FUNCTION_BLOCK FINAL FB_Tilt_A EXTENDS FB_StatusExecuteFB
VAR_IN_OUT
	fbMover								: MC_PlanarMover;
END_VAR
VAR_INPUT
	Execute								: BOOL;
	Position							: ST_POSITION;
	Velocity							: LREAL;
	Acceleration						: LREAL;
	Deceleration						: LREAL;
	Jerk								: LREAL;
END_VAR
VAR_OUTPUT
	Done								: BOOL;
	Busy								: BOOL;
	CommandAborted						: BOOL;
	Error								: BOOL;
	ErrorID								: UDINT;
END_VAR
VAR
	uiState								: UINT;
	//Input 内部変数
	dutPosition							: ST_POSITION;
	lrVelocity							: LREAL;
	lrAcceleration						: LREAL;
	lrDeceleration						: LREAL;
	lrJerk								: LREAL;
	
	//ローカル
	fbFB_Mover							: MC_PlanarFeedback;
	dutTargetPosition					: ST_POSITION;
	fbConstraint						: DynamicConstraint_PathXY;
	fbMoveA								: FB_MoveA;
END_VAR

Prop_Execute := Execute;
METH_Main();

fbFB_Mover.Update();

Busy := bBusy;
Done := bDone;
CommandAborted := bCommandAborted;
Error := bError;
ErrorID := udiErrorID;

//{error 'add method implementation or delete method to use base implementation'}
METHOD INTERNAL METH_Busy : BOOL
IF fbFB_Mover.Error THEN
	METH_Error();
	Prop_ErrorID := fbFB_Mover.ErrorId; //Moverがエラー
	RETURN;
END_IF
IF THIS^.fbMover.MCTOPLC.STD.State = MC_PLANAR_STATE.Error THEN
	METH_Error();
	Prop_ErrorID := 1; //Moverがエラー
	RETURN;
END_IF
IF fbFB_Mover.Aborted THEN
	METH_CommandAborted();
	RETURN;
END_IF

CASE THIS^.uiState OF
	0:
	//+Aに傾ける
	dutTargetPosition.a := dutPosition.a;
	fbMoveA(
		fbMover:= THIS^.fbMover, 
		Execute:= TRUE, 
		Position:= dutTargetPosition, 
		Velocity:= THIS^.lrVelocity, 
		Acceleration:= THIS^.lrAcceleration, 
		Deceleration:= THIS^.lrDeceleration, 
		Jerk:= THIS^.lrJerk);
	IF fbMoveA.Done THEN
		fbMoveA(fbMover:= THIS^.fbMover, Execute:= FALSE);
		THIS^.uiState := 10;
	ELSIF fbMoveA.Error THEN
		METH_Error();
		Prop_ErrorID := 10; //Moverがエラー
	END_IF
	
	10:
	//-Aに傾ける
	dutTargetPosition.a := -1*dutPosition.a;
	fbMoveA(
		fbMover:= THIS^.fbMover, 
		Execute:= TRUE, 
		Position:= dutTargetPosition, 
		Velocity:= THIS^.lrVelocity, 
		Acceleration:= THIS^.lrAcceleration, 
		Deceleration:= THIS^.lrDeceleration, 
		Jerk:= THIS^.lrJerk);
	IF fbMoveA.Done THEN
		fbMoveA(fbMover:= THIS^.fbMover, Execute:= FALSE);
		THIS^.uiState := 30;
	ELSIF fbMoveA.Error THEN
		METH_Error();
		Prop_ErrorID := 11; //Moverがエラー
	END_IF

	30:
	//0に戻す
	dutTargetPosition.a := 0;
	fbMoveA(
		fbMover:= THIS^.fbMover, 
		Execute:= TRUE, 
		Position:= dutTargetPosition, 
		Velocity:= THIS^.lrVelocity, 
		Acceleration:= THIS^.lrAcceleration, 
		Deceleration:= THIS^.lrDeceleration, 
		Jerk:= THIS^.lrJerk);
	IF fbMoveA.Done THEN
		fbMoveA(fbMover:= THIS^.fbMover, Execute:= FALSE);
		THIS^.uiState := 16#FFFF;
	ELSIF fbMoveA.Error THEN
		METH_Error();
		Prop_ErrorID := 12; //Moverがエラー
	END_IF
	
	16#FFFF:
	METH_Done();
END_CASE
END_METHOD

 {attribute 'hide'}
//{error 'add method implementation or delete method to use base implementation'}
METHOD INTERNAL METH_Enter : BOOL
//Input 内部変数に移す
dutPosition := Position;
lrVelocity := Velocity;
lrAcceleration := Acceleration;
lrDeceleration := Deceleration;
lrJerk := Jerk;
END_METHOD

 {attribute 'hide'}
//{error 'add method implementation or delete method to use base implementation'}
METHOD INTERNAL METH_Exit : BOOL
Prop_Done := FALSE;
Prop_Busy := FALSE;
Prop_CommandAborted := FALSE;
Prop_Error := FALSE;
Prop_ErrorID := 0;

// 内部変数をリフレッシュする
uiState := 0;
lrVelocity := 0;
lrAcceleration := 0;
lrDeceleration := 0;
lrJerk := 0;

//FBの初期化
fbMoveA(fbMover:= THIS^.fbMover, Execute:= FALSE);
END_METHOD

 {attribute 'hide'}
//{error 'add method implementation or delete method to use base implementation'}
METHOD INTERNAL METH_Main : BOOL
//Doneに遷移
IF SUPER^.bDone AND SUPER^.bExecute THEN
	METH_Done();
	RETURN;
END_IF
//Errorに遷移
IF SUPER^.bError AND SUPER^.bExecute THEN
	METH_Error();
	RETURN;
END_IF
//CommandAbortedに遷移
IF SUPER^.bCommandAborted AND SUPER^.bExecute THEN
	METH_CommandAborted();
	RETURN;
END_IF
//FBをリフレッシュ
//状態がDone, Error, CommandAborted時に Execute FALSE で遷移
IF (SUPER^.bDone OR SUPER^.bError OR SUPER^.bCommandAborted) AND NOT SUPER^.bExecute THEN
	METH_Exit();
	RETURN;
END_IF

//実行開始
IF SUPER^.bExecute AND NOT SUPER^.bBusy THEN
	METH_Execute();
	METH_Enter();
END_IF
//実行中
IF SUPER^.bBusy THEN
	METH_Busy();
END_IF
END_METHOD

END_FUNCTION_BLOCK

(* stored: Version 1.1.0.1, ProductVersion 3.1.4024.12
   POU FB_Tilt_A: Id {db625dc9-5fd0-45ad-b494-67861582e8f8}, SpecialFunc None
   Method METH_Busy: Id {9ff795b3-3cce-4732-9bca-9b032c9aea48}
   Method METH_Enter: Id {40e40d96-2c5f-497b-8347-c374bcee5f5a}
   Method METH_Exit: Id {6ed1c824-1fb3-498e-9d48-02133266c88c}
   Method METH_Main: Id {d792ff9e-0de0-4a05-8e41-3f003cfd5ff8} *)
